// TIA Portal project "FactoryIO_Template_S7-1200_V16_V16" (V16)
// Vorlageprojekt für das Buch mit Zielsystem S7-1200

(* hardware
DEVICE "S7-1200-Station_1"  S7-1200 Station
   slot 0: "Baugruppenträger_0"  Rack  V1.0
   slot 1: "PLC_1"  CPU 1211C DC/DC/DC  6ES7 211-1AE40-0XB0  V4.1
*)

// ===== PLC "PLC_1"  CPU 1211C DC/DC/DC =====

VAR_GLOBAL   // PLC tag table "Standard-Variablentabelle"
   "belt 1" AT %A0.0 : Bool;
   "start" AT %E0.0 : Bool;
   "stop" AT %E0.1 : Bool;
   "Tag_4" AT %I10.0 : Bool;
   "Tag_5" AT %Q10.0 : Bool;
   "Tag_6" AT %I10.1 : Bool;
   "x" AT %M0.0 : Bool;
   "belt 2" AT %Q0.1 : Bool;
   "belt 3" AT %Q0.2 : Bool;
   "back limit" AT %I0.2 : Bool;
   "roller +" AT %Q0.3 : Bool;
   "Tag_1" AT %M0.1 : Bool;
   "diffuse sensor 4" AT %I0.3 : Bool;
   "front limit" AT %I0.4 : Bool;
   "turntable 1 turn" AT %Q0.4 : Bool;
   "limit 90" AT %I0.5 : Bool;
   "diffuse sensor 1" AT %I0.6 : Bool;
   "diffuse sensor 3" AT %I0.7 : Bool;
   "limit 0" AT %I1.0 : Bool;
   "roller -" AT %Q0.5 : Bool;
END_VAR

// folder: System blocks/Program resources

DATA_BLOCK "C1"   // DB1
{ S7_Optimized_Access := 'TRUE' }
AUTHOR : Simatic
FAMILY : IEC
NAME : CNTR
VERSION : 1.0
// stored: InstanceOfName IEC_COUNTER
"IEC_COUNTER"
BEGIN
END_DATA_BLOCK

DATA_BLOCK "T1"   // DB2
{ S7_Optimized_Access := 'TRUE' }
AUTHOR : Simatic
FAMILY : IEC
NAME : IEC_TMR
VERSION : 1.0
// stored: InstanceOfName IEC_TIMER
"IEC_TIMER"
BEGIN
END_DATA_BLOCK

// folder: (top level)

FUNCTION "MHJ-PLC-Lab-Function-S71200" : Void   // FC9000, SCL
{ S7_Optimized_Access := 'TRUE' }
VERSION : 0.1
   VAR_TEMP
      rdTimeReturn : Int;
      outputTime : DTL;
      SyncVal : Byte;
      forVal : Int;
      forVal_2 : Int;
      Value : Byte;
   END_VAR
   VAR CONSTANT
      CompVal : Byte := 16#34;
      Value_01 : Byte := 16#11;
      Value_01_DW : DWord := 16#A165_D992;
      Value_02_DW : DWord := 16#58BE_4401;
   END_VAR
BEGIN

   #Value:=PEEK(area := 16#82,
        dbNumber := 0,
        byteOffset := 511);
   #Value := #Value + 1;

   POKE(area := 16#82,
        dbNumber := 0,
        byteOffset := 511,
        value := #Value);

   POKE(area:=16#81,
        dbNumber:=0,
        byteOffset:=1016,
        value:=#Value_01_DW);
   POKE(area := 16#81,
        dbNumber := 0,
        byteOffset := 1020,
        value := #Value_02_DW);

   POKE(area := 16#81,
        dbNumber := 0,
        byteOffset := 511,
        value := B#16#00);

   FOR #forVal := 0 TO 120 DO
       FOR #forVal_2:=0 TO 10 DO
           #rdTimeReturn:=RD_SYS_T(#outputTime);
           #rdTimeReturn := WR_SYS_T(#outputTime);
           #rdTimeReturn := RD_SYS_T(#outputTime);
           #rdTimeReturn := WR_SYS_T(#outputTime);
       END_FOR;
       #SyncVal:= PEEK(area := 16#81,
                      dbNumber := 0,
                      byteOffset := 511);
       IF #SyncVal = #CompVal THEN
          GOTO M_1;
       END_IF;
   END_FOR;
   RETURN;

   M_1:
   POKE(area := 16#81,
        dbNumber := 0,
        byteOffset := 511,
        value := B#16#0);
END_FUNCTION

ORGANIZATION_BLOCK "Main"   // OB1, LAD, ProgramCycle
TITLE = "Main Program Sweep (Cycle)"
{ S7_Optimized_Access := 'TRUE' }
VERSION : 0.1
   VAR_INPUT
      Initial_Call : Bool;   // Initial call of this OB
      Remanence : Bool;   // =True, if remanent data are available
   END_VAR
   VAR_TEMP   // added for the SCL form of the ladder/FBD networks
      _w1 : Bool;
   END_VAR
BEGIN

REGION Network 1: Konnektierungsbaustein für PLC-Lab
   // Im Netzwerk 1 wird der Konnektierungsbaustein für PLC-Lab aufgerufen.
   // Dieser Aufruf darf nicht entfernt werden!
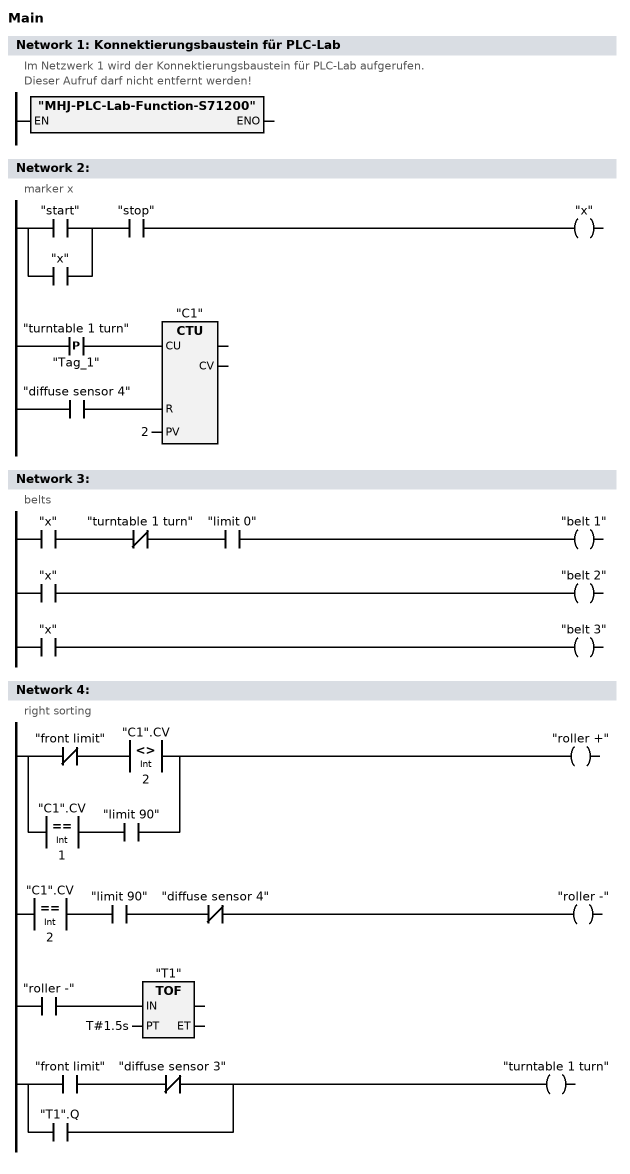
   RUNG wire#powerrail
      "MHJ-PLC-Lab-Function-S71200"()
   END_RUNG
   // the same network as SCL:
   "MHJ-PLC-Lab-Function-S71200"();
END_REGION

REGION Network 2
   // marker x
   "x" := ("start" OR "x") AND "stop";
   #_w1 := "turntable 1 turn" AND NOT "Tag_1";   // rising edge of "turntable 1 turn"
   "Tag_1" := "turntable 1 turn";
   "C1".CTU(CU := #_w1, R := "diffuse sensor 4", PV := 2);
END_REGION

REGION Network 3
   // belts
   RUNG wire#powerrail
      Contact( "x" )
      I_Contact( "turntable 1 turn" )
      Contact( "limit 0" )
      Coil( "belt 1" )
   END_RUNG
   RUNG wire#powerrail
      Contact( "x" )
      Coil( "belt 2" )
   END_RUNG
   RUNG wire#powerrail
      Contact( "x" )
      Coil( "belt 3" )
   END_RUNG
   // the same network as SCL:
   "belt 1" := "x" AND NOT "turntable 1 turn" AND "limit 0";
   "belt 2" := "x";
   "belt 3" := "x";
END_REGION

REGION Network 4
   // right sorting
   "roller +" := (NOT "front limit" AND ("C1".CV <> 2)) OR (("C1".CV = 1) AND "limit 90");
   "roller -" := ("C1".CV = 2) AND "limit 90" AND NOT "diffuse sensor 4";
   "T1".TOF(IN := "roller -", PT := T#1.5s);
   "turntable 1 turn" := ("front limit" AND NOT "diffuse sensor 3") OR "T1".Q;
END_REGION
END_ORGANIZATION_BLOCK